INTERFACE I_CYLINDER_SA_GENERAL EXTENDS I_GENERAL_OBJECT

METHOD M_PressureCalibration : BOOL
VAR_INPUT
END_VAR
END_METHOD

METHOD M_Reset : BOOL
VAR_INPUT
END_VAR
END_METHOD

METHOD M_SetReady : BOOL
VAR_INPUT
END_VAR
END_METHOD

METHOD M_SetWorkPressure : BOOL
VAR_INPUT
  ePressureType:                   E_PRESSURE_TYPE;
  rWorkPressure:                   REAL;
END_VAR
END_METHOD

METHOD M_SetWorkPressureZero : BOOL
VAR_INPUT
END_VAR
END_METHOD

METHOD M_Stop : BOOL
VAR_INPUT
END_VAR
END_METHOD

METHOD M_ToWP : BOOL
VAR_INPUT
  /// Bar | Force in N | Percent 0-100 | Value 0-32767
  ePressureType:            E_PRESSURE_TYPE;
  rWorkPressure:            REAL;
  bPressureRegulation:      BOOL;
  /// Just need for prop valve
  eSpeedType:               E_SPEED_TYPE;
  rSpeed:                   REAL;
END_VAR
END_METHOD

PROPERTY P_CurrentForceInKN : REAL
GET
END_GET
END_PROPERTY

PROPERTY P_PistonSurfaceA : LREAL
GET
END_GET
END_PROPERTY

PROPERTY P_PressureOk : BOOL
GET
END_GET
END_PROPERTY

PROPERTY P_ReadyState : BOOL
GET
END_GET
END_PROPERTY

PROPERTY P_WorkPressure : REAL
GET
END_GET
END_PROPERTY

END_INTERFACE

(* stored: Version 1.1.0.1, ProductVersion 3.1.4024.12
   Itf I_CYLINDER_SA_GENERAL: Id {13805b17-5bfc-449b-bce9-c48e9afa8a30}
   Method M_PressureCalibration: Id {3207f34c-227e-4e34-88d0-061c2a3c0606}
   Method M_Reset: Id {63bd97a7-dbf3-4709-b6ed-12bdf42f2c1a}
   Method M_SetReady: Id {526e01c0-25c3-4f5d-9c5d-118de864d5ca}
   Method M_SetWorkPressure: Id {27b87d49-3fa1-4e2b-87c0-4c8d66261cea}
   Method M_SetWorkPressureZero: Id {d0043780-b8ba-4d47-a388-09297da08fc8}
   Method M_Stop: Id {5d16f8e8-c647-4b76-ab9b-0e37bc939372}
   Method M_ToWP: Id {9f93042e-6a04-4402-8079-5bcf67d76e66}
   Property P_CurrentForceInKN: Id {38779810-f63e-40d5-ad5a-d486b1bf9973}
   Get Get: Id {1202eba7-fd5e-4b0f-bead-b2451cba5f27}
   Property P_PistonSurfaceA: Id {cb7a7031-d80b-4299-86ba-083abc5221df}
   Get Get: Id {4e13b714-5fd6-4130-a212-ab2c3c8e985c}
   Property P_PressureOk: Id {dd264b0b-600d-4fda-b8ab-fc785f881925}
   Get Get: Id {6d65a202-d413-4f0f-baa3-711fa2c85d81}
   Property P_ReadyState: Id {0740d98d-e1ea-4a26-b0ca-7196aec5a971}
   Get Get: Id {83b47822-94f4-4930-95fb-53eb1264c36c}
   Property P_WorkPressure: Id {e1a33b87-7f65-4ff6-a069-934218d97fa5}
   Get Get: Id {912e89bc-bdc3-4d4f-bad4-d21fda373182} *)
